(* Gets the upper bound index of :itf:`I_Runnable` array.*)
FUNCTION F_GetRunnableArrayUpperBound : T_Position
VAR_IN_OUT
	arRunnables : ARRAY[*] OF REAL; // The array to query.
END_VAR

F_GetRunnableArrayUpperBound := LOWER_BOUND(arRunnables, 1);

END_FUNCTION

(* stored: Version 1.1.0.1
   POU F_GetRunnableArrayUpperBound: Id {276aef35-628c-0a75-27c5-ad6a6b5c0cd9}, SpecialFunc None *)
